# EPICS autosave request: measCompApp/Db/C9513_module_settings.req
$(P)$(R)BoWord
